// TIA Portal V21 export
TYPE "Std_TCiclo"
   STRUCT
      Act : LReal;   // Attuale
      PercTciclo : Real;   // Percentuale tempo ciclo utilizzato
   END_STRUCT;
END_TYPE
